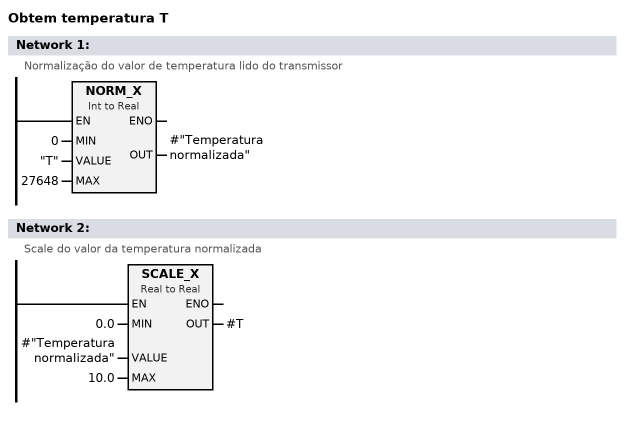
   RUNG wire#powerrail
      { S7_Templates := "[SrcType := Int, DestType := Real]" } Normalize(min := 0, value := "T", max := 27648, out => #"Temperatura normalizada")
   END_RUNG
   // the same network as SCL:
   #"Temperatura normalizada" := NORM_X(MIN := 0, VALUE := "T", MAX := 27648);
END_REGION

REGION Network 2
   // Scale do valor da temperatura normalizada
   RUNG wire#powerrail
      { S7_Templates := "[SrcType := Real, DestType := Real]" } Scale(min := 0.0, value := #"Temperatura normalizada", max := 10.0, out => #T)
   END_RUNG
   // the same network as SCL:
   #T := SCALE_X(MIN := 0.0, VALUE := #"Temperatura normalizada", MAX := 10.0);
END_REGION
END_FUNCTION

FUNCTION "Obtem temperatura TA" : Void   // FC23, LAD
{ S7_Optimized_Access := 'TRUE' }
VERSION : 0.1
   VAR_OUTPUT
      TA : Real;   // Temperatura obtida
   END_VAR
   VAR_TEMP
      "Temperatura normalizada" : Real;   // Temperatura normalizada
   END_VAR
BEGIN

REGION Network 1
   // Normalização do valor de temperatura lido do transmissor
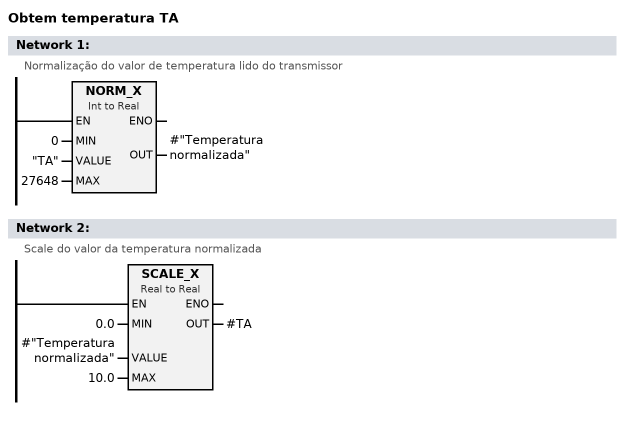
   RUNG wire#powerrail
      { S7_Templates := "[SrcType := Int, DestType := Real]" } Normalize(min := 0, value := "TA", max := 27648, out => #"Temperatura normalizada")
   END_RUNG
   // the same network as SCL:
   #"Temperatura normalizada" := NORM_X(MIN := 0, VALUE := "TA", MAX := 27648);
END_REGION

REGION Network 2
   // Scale do valor da temperatura normalizada
   RUNG wire#powerrail
      { S7_Templates := "[SrcType := Real, DestType := Real]" } Scale(min := 0.0, value := #"Temperatura normalizada", max := 10.0, out => #TA)
   END_RUNG
   // the same network as SCL:
   #TA := SCALE_X(MIN := 0.0, VALUE := #"Temperatura normalizada", MAX := 10.0);
END_REGION
END_FUNCTION

FUNCTION "Aciona VD2" : Void   // FC24, LAD
{ S7_Optimized_Access := 'TRUE' }
VERSION : 0.1
BEGIN

REGION Network 1: Válvula on/off da linha direta (segunda)
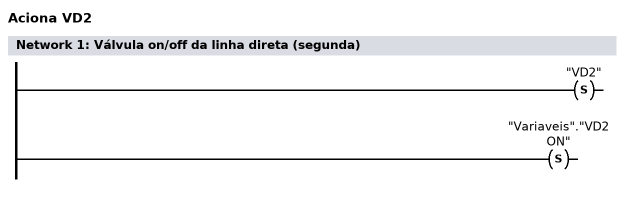
   RUNG wire#powerrail
      S_Coil( "VD2" )
   END_RUNG
   RUNG wire#powerrail
      S_Coil( "Variaveis"."VD2 ON" )
   END_RUNG
   // the same network as SCL:
   "VD2" := TRUE;
   "Variaveis"."VD2 ON" := TRUE;
END_REGION
END_FUNCTION

FUNCTION "Desliga VD2" : Void   // FC25, LAD
{ S7_Optimized_Access := 'TRUE' }
VERSION : 0.1
BEGIN

REGION Network 1: Válvula on/off da linha direta (segunda)
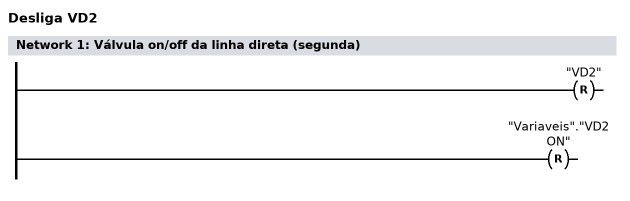
   RUNG wire#powerrail
      R_Coil( "VD2" )
   END_RUNG
   RUNG wire#powerrail
      R_Coil( "Variaveis"."VD2 ON" )
   END_RUNG
   // the same network as SCL:
   "VD2" := FALSE;
   "Variaveis"."VD2 ON" := FALSE;
END_REGION
END_FUNCTION

FUNCTION "Etapa pausada" : Void   // FC26, LAD
{ S7_Optimized_Access := 'TRUE' }
VERSION : 0.1
   VAR_TEMP   // added for the SCL form of the ladder/FBD networks
      _w1 : Bool;
      _w2 : Bool;
   END_VAR
BEGIN

REGION Network 1: LED que indica o estado de etapa pausada
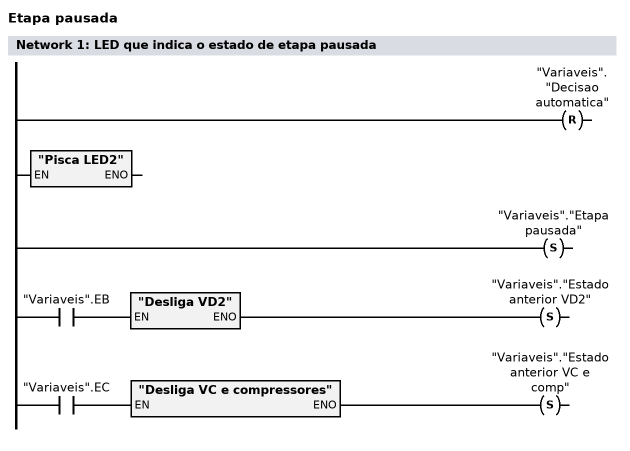
   RUNG wire#powerrail
      R_Coil( "Variaveis"."Decisao automatica" )
   END_RUNG
   RUNG wire#powerrail
      "Pisca LED2"()
   END_RUNG
   RUNG wire#powerrail
      S_Coil( "Variaveis"."Etapa pausada" )
   END_RUNG
   RUNG wire#powerrail
      Contact( "Variaveis".EB )
      "Desliga VD2"()
      S_Coil( "Variaveis"."Estado anterior VD2" )
   END_RUNG
   RUNG wire#powerrail
      Contact( "Variaveis".EC )
      "Desliga VC e compressores"()
      S_Coil( "Variaveis"."Estado anterior VC e comp" )
   END_RUNG
   // the same network as SCL:
   "Variaveis"."Decisao automatica" := FALSE;
   "Pisca LED2"();
   "Variaveis"."Etapa pausada" := TRUE;
   "Desliga VD2"(EN := "Variaveis".EB, ENO => #_w1);
   IF #_w1 THEN "Variaveis"."Estado anterior VD2" := TRUE; END_IF;
   "Desliga VC e compressores"(EN := "Variaveis".EC, ENO => #_w2);
   IF #_w2 THEN "Variaveis"."Estado anterior VC e comp" := TRUE; END_IF;
END_REGION
END_FUNCTION

FUNCTION "Etapa retomada" : Void   // FC27, LAD
{ S7_Optimized_Access := 'TRUE' }
VERSION : 0.1
BEGIN

REGION Network 1: LED que indica o estado de etapa pausada
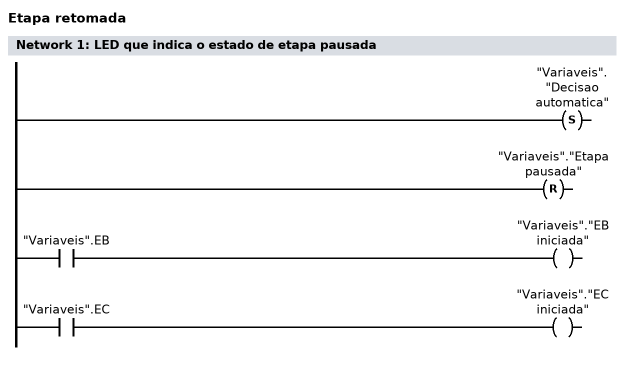
   RUNG wire#powerrail
      S_Coil( "Variaveis"."Decisao automatica" )
   END_RUNG
   RUNG wire#powerrail
      R_Coil( "Variaveis"."Etapa pausada" )
   END_RUNG
   RUNG wire#powerrail
      Contact( "Variaveis".EB )
      Coil( "Variaveis"."EB iniciada" )
   END_RUNG
   RUNG wire#powerrail
      Contact( "Variaveis".EC )
      Coil( "Variaveis"."EC iniciada" )
   END_RUNG
   // the same network as SCL:
   "Variaveis"."Decisao automatica" := TRUE;
   "Variaveis"."Etapa pausada" := FALSE;
   "Variaveis"."EB iniciada" := "Variaveis".EB;
   "Variaveis"."EC iniciada" := "Variaveis".EC;
END_REGION
END_FUNCTION

FUNCTION "Verifica VC 1" : Void   // FC28, LAD
{ S7_Optimized_Access := 'TRUE' }
VERSION : 0.1
BEGIN

REGION Network 1: Válvula on/off da entrada do sistema de compressores
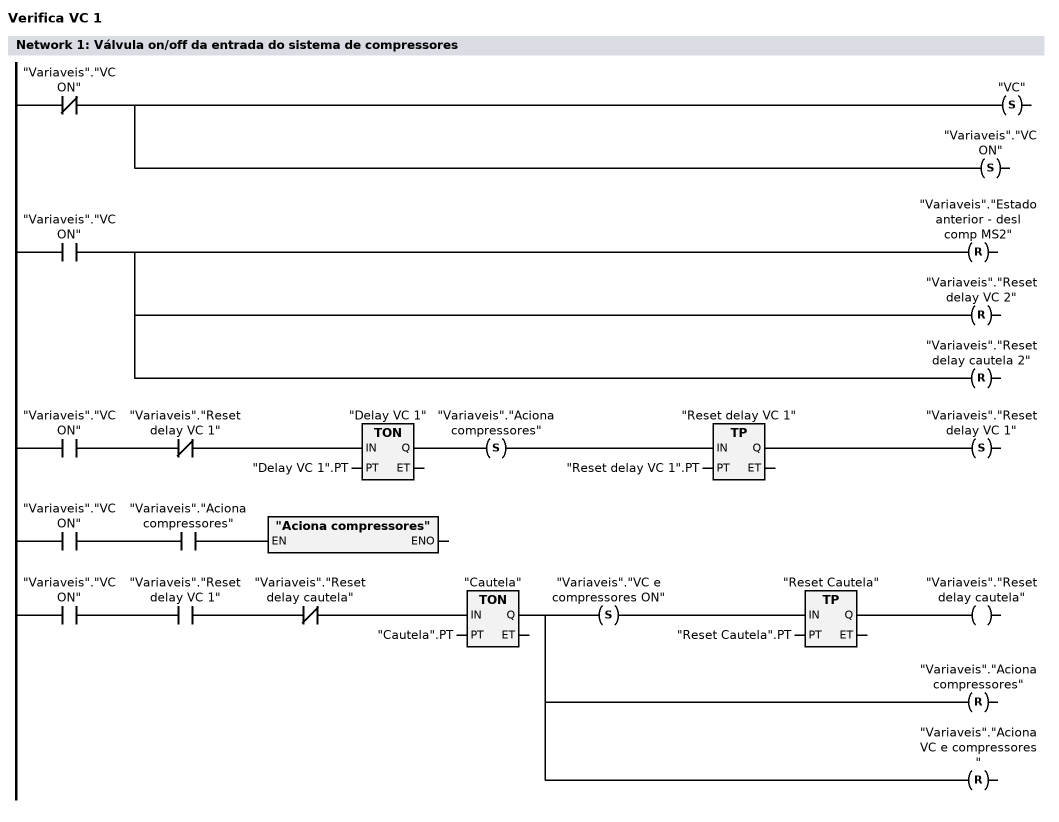
   IF NOT "Variaveis"."VC ON" THEN
       "VC" := TRUE;
       "Variaveis"."VC ON" := TRUE;
   END_IF;
   IF "Variaveis"."VC ON" THEN
       "Variaveis"."Estado anterior - desl comp MS2" := FALSE;
       "Variaveis"."Reset delay VC 2" := FALSE;
       "Variaveis"."Reset delay cautela 2" := FALSE;
   END_IF;
   "Delay VC 1".TON(IN := "Variaveis"."VC ON" AND NOT "Variaveis"."Reset delay VC 1", PT := "Delay VC 1".PT);
   IF "Delay VC 1".Q THEN "Variaveis"."Aciona compressores" := TRUE; END_IF;
   "Reset delay VC 1".TP(IN := "Delay VC 1".Q, PT := "Reset delay VC 1".PT);
   IF "Reset delay VC 1".Q THEN "Variaveis"."Reset delay VC 1" := TRUE; END_IF;
   IF "Variaveis"."VC ON" AND "Variaveis"."Aciona compressores" THEN "Aciona compressores"(); END_IF;
   "Cautela".TON(IN := "Variaveis"."VC ON" AND "Variaveis"."Reset delay VC 1" AND NOT "Variaveis"."Reset delay cautela",
                 PT := "Cautela".PT);
   IF "Cautela".Q THEN "Variaveis"."VC e compressores ON" := TRUE; END_IF;
   "Reset Cautela".TP(IN := "Cautela".Q, PT := "Reset Cautela".PT);
   "Variaveis"."Reset delay cautela" := "Reset Cautela".Q;
   IF "Cautela".Q THEN
       "Variaveis"."Aciona compressores" := FALSE;
       "Variaveis"."Aciona VC e compressores" := FALSE;
   END_IF;
END_REGION
END_FUNCTION

FUNCTION "Verifica VC 2" : Void   // FC29, LAD
{ S7_Optimized_Access := 'TRUE' }
VERSION : 0.1
BEGIN

REGION Network 1: Válvula on/off da entrada do sistema de compressores
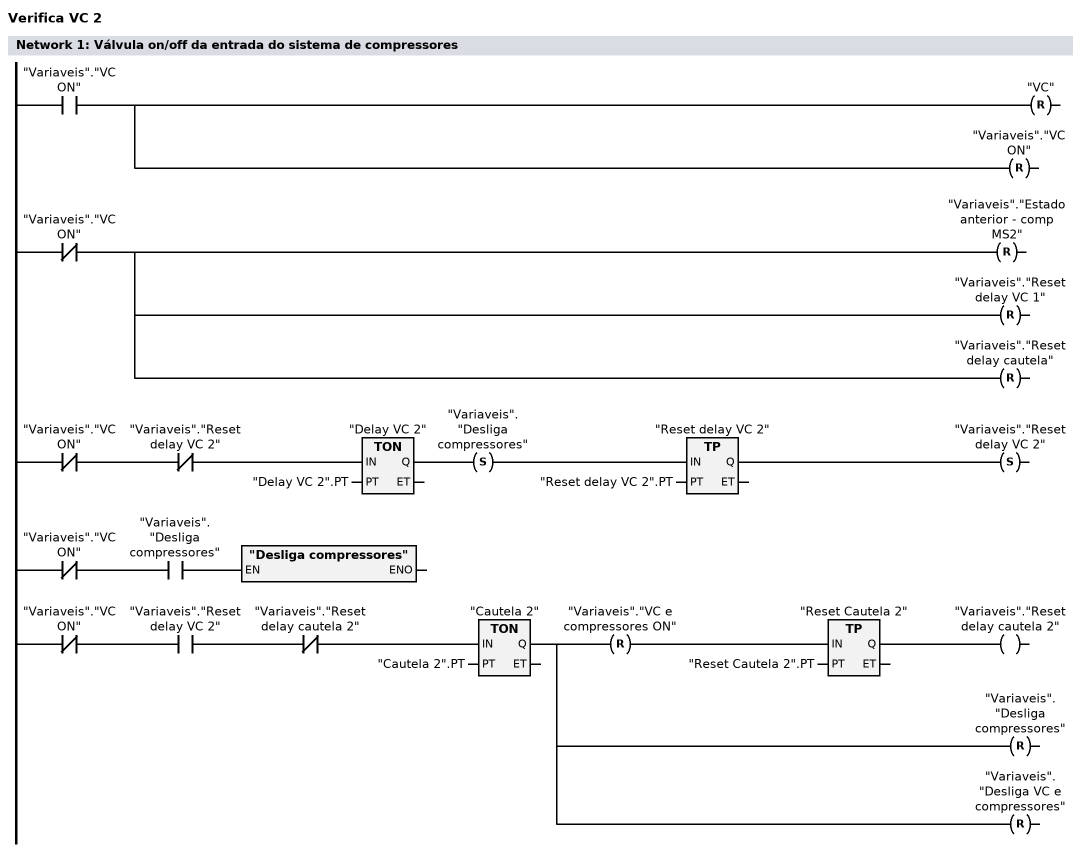
   IF "Variaveis"."VC ON" THEN
       "VC" := FALSE;
       "Variaveis"."VC ON" := FALSE;
   END_IF;
   IF NOT "Variaveis"."VC ON" THEN
       "Variaveis"."Estado anterior - comp MS2" := FALSE;
       "Variaveis"."Reset delay VC 1" := FALSE;
       "Variaveis"."Reset delay cautela" := FALSE;
   END_IF;
   "Delay VC 2".TON(IN := NOT "Variaveis"."VC ON" AND NOT "Variaveis"."Reset delay VC 2", PT := "Delay VC 2".PT);
   IF "Delay VC 2".Q THEN "Variaveis"."Desliga compressores" := TRUE; END_IF;
   "Reset delay VC 2".TP(IN := "Delay VC 2".Q, PT := "Reset delay VC 2".PT);
   IF "Reset delay VC 2".Q THEN "Variaveis"."Reset delay VC 2" := TRUE; END_IF;
   IF NOT "Variaveis"."VC ON" AND "Variaveis"."Desliga compressores" THEN "Desliga compressores"(); END_IF;
   "Cautela 2".TON(IN := NOT "Variaveis"."VC ON" AND "Variaveis"."Reset delay VC 2" AND NOT "Variaveis"."Reset delay cautela 2",
                   PT := "Cautela 2".PT);
   IF "Cautela 2".Q THEN "Variaveis"."VC e compressores ON" := FALSE; END_IF;
   "Reset Cautela 2".TP(IN := "Cautela 2".Q, PT := "Reset Cautela 2".PT);
   "Variaveis"."Reset delay cautela 2" := "Reset Cautela 2".Q;
   IF "Cautela 2".Q THEN
       "Variaveis"."Desliga compressores" := FALSE;
       "Variaveis"."Desliga VC e compressores" := FALSE;
   END_IF;
END_REGION
END_FUNCTION

FUNCTION "Aciona VC e compressores" : Void   // FC30, LAD
{ S7_Optimized_Access := 'TRUE' }
VERSION : 0.1
BEGIN

REGION Network 1
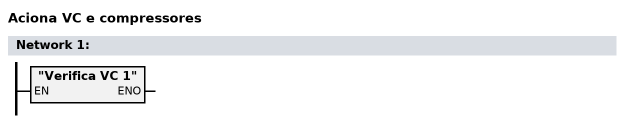
   RUNG wire#powerrail
      "Verifica VC 1"()
   END_RUNG
   // the same network as SCL:
   "Verifica VC 1"();
END_REGION
END_FUNCTION

FUNCTION "Desliga VC e compressores" : Void   // FC31, LAD
{ S7_Optimized_Access := 'TRUE' }
VERSION : 0.1
BEGIN

REGION Network 1
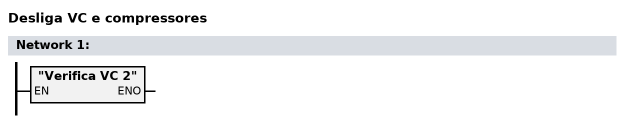
   RUNG wire#powerrail
      "Verifica VC 2"()
   END_RUNG
   // the same network as SCL:
   "Verifica VC 2"();
END_REGION
END_FUNCTION

FUNCTION "EB - Etapa iniciada" : Void   // FC32, LAD
{ S7_Optimized_Access := 'TRUE' }
VERSION : 0.1
   VAR_TEMP
      T : Real;   // Temperatura no nó estendido
      TA : Real;   // Temperatura ambiente
      PN : Real;   // Pressão no nó estendido
      PSF6 : Real;   // Pressão do tanque de SF6
      "Threshold ambiente" : Real;   // (1 - beta)*TA
      "Threshold PSF6" : Real;   // (1 + gamma)*PSF6
   END_VAR
   VAR_TEMP   // added for the SCL form of the ladder/FBD networks
      _w1 : Bool;
      _w2 : Bool;
      _w3 : Bool;
      _w4 : Bool;
   END_VAR
BEGIN

REGION Network 1
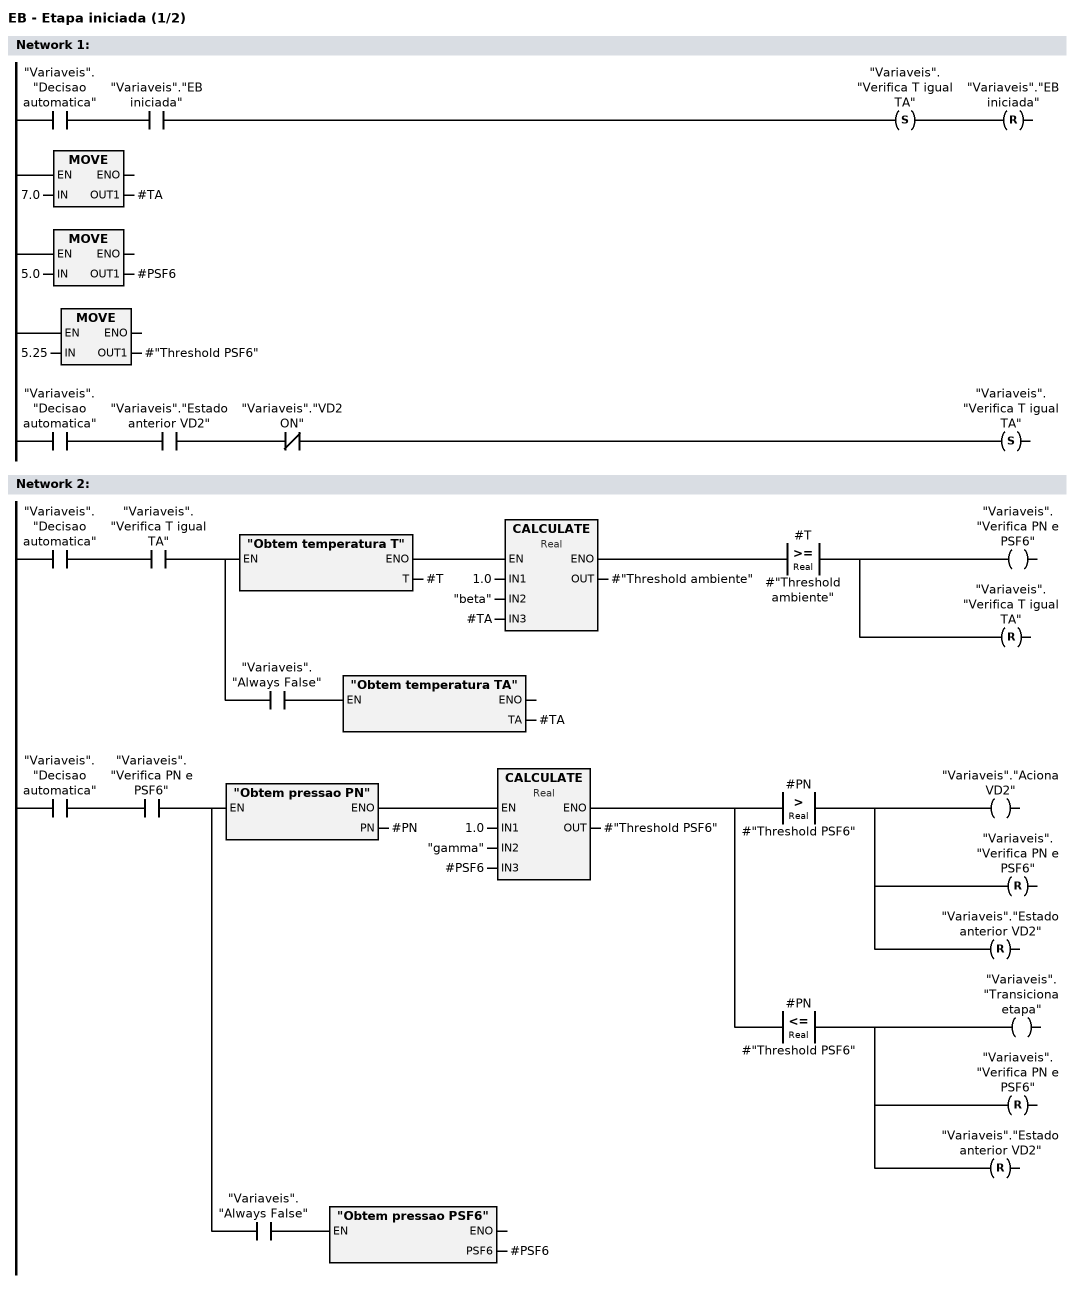
   RUNG wire#powerrail
      Contact( "Variaveis"."Decisao automatica" )
      Contact( "Variaveis"."EB iniciada" )
      S_Coil( "Variaveis"."Verifica T igual TA" )
      R_Coil( "Variaveis"."EB iniciada" )
   END_RUNG
   RUNG wire#powerrail
      Move(in := 7.0, out1 => #TA)
   END_RUNG
   RUNG wire#powerrail
      Move(in := 5.0, out1 => #PSF6)
   END_RUNG
   RUNG wire#powerrail
      Move(in := 5.25, out1 => #"Threshold PSF6")
   END_RUNG
   RUNG wire#powerrail
      Contact( "Variaveis"."Decisao automatica" )
      Contact( "Variaveis"."Estado anterior VD2" )
      I_Contact( "Variaveis"."VD2 ON" )
      S_Coil( "Variaveis"."Verifica T igual TA" )
   END_RUNG
   // the same network as SCL:
   IF "Variaveis"."Decisao automatica" AND "Variaveis"."EB iniciada" THEN
       "Variaveis"."Verifica T igual TA" := TRUE;
       "Variaveis"."EB iniciada" := FALSE;
   END_IF;
   #TA := 7.0;
   #PSF6 := 5.0;
   #"Threshold PSF6" := 5.25;
   IF "Variaveis"."Decisao automatica" AND "Variaveis"."Estado anterior VD2" AND NOT "Variaveis"."VD2 ON" THEN
       "Variaveis"."Verifica T igual TA" := TRUE;
   END_IF;
END_REGION

REGION Network 2
   RUNG wire#powerrail
      Contact( "Variaveis"."Decisao automatica" )
      Contact( "Variaveis"."Verifica T igual TA" )
      wire#w1
      "Obtem temperatura T"(T => #T)
      { S7_Templates := "SrcType := Real"; S7_Expression := "(IN1 - IN2) * IN3" } Calculate(in1 := 1.0, in2 := "beta", in3 := #TA, out => #"Threshold ambiente")
      { S7_Templates := "SrcType := Real" } GE_Contact(in1 := #T, in2 := #"Threshold ambiente")
      wire#w2
      Coil( "Variaveis"."Verifica PN e PSF6" )
   END_RUNG
   RUNG wire#w2
      R_Coil( "Variaveis"."Verifica T igual TA" )
   END_RUNG
   RUNG wire#w1
      Contact( "Variaveis"."Always False" )
      "Obtem temperatura TA"(TA => #TA)
   END_RUNG
   RUNG wire#powerrail
      Contact( "Variaveis"."Decisao automatica" )
      Contact( "Variaveis"."Verifica PN e PSF6" )
      wire#w3
      "Obtem pressao PN"(PN => #PN)
      { S7_Templates := "SrcType := Real"; S7_Expression := "(IN1 + IN2) * IN3" } Calculate(in1 := 1.0, in2 := "gamma", in3 := #PSF6, out => #"Threshold PSF6")
      wire#w4
      { S7_Templates := "SrcType := Real" } GT_Contact(in1 := #PN, in2 := #"Threshold PSF6")
      wire#w5
      Coil( "Variaveis"."Aciona VD2" )
   END_RUNG
   RUNG wire#w5
      R_Coil( "Variaveis"."Verifica PN e PSF6" )
   END_RUNG
   RUNG wire#w5
      R_Coil( "Variaveis"."Estado anterior VD2" )
   END_RUNG
   RUNG wire#w4
      { S7_Templates := "SrcType := Real" } LE_Contact(in1 := #PN, in2 := #"Threshold PSF6")
      wire#w6
      Coil( "Variaveis"."Transiciona etapa" )
   END_RUNG
   RUNG wire#w6
      R_Coil( "Variaveis"."Verifica PN e PSF6" )
   END_RUNG
   RUNG wire#w6
      R_Coil( "Variaveis"."Estado anterior VD2" )
   END_RUNG
   RUNG wire#w3
      Contact( "Variaveis"."Always False" )
      "Obtem pressao PSF6"(PSF6 => #PSF6)
   END_RUNG
   // the same network as SCL:
   #_w1 := "Variaveis"."Decisao automatica" AND "Variaveis"."Verifica T igual TA";
   "Obtem temperatura T"(EN := #_w1, T => #T, ENO => #_w2);
   IF #_w2 THEN #"Threshold ambiente" := (1.0 - "beta") * #TA; END_IF;
   "Variaveis"."Verifica PN e PSF6" := #_w2 AND (#T >= #"Threshold ambiente");
   IF "Variaveis"."Verifica PN e PSF6" THEN "Variaveis"."Verifica T igual TA" := FALSE; END_IF;
   IF #_w1 AND "Variaveis"."Always False" THEN "Obtem temperatura TA"(TA => #TA); END_IF;
   #_w3 := "Variaveis"."Decisao automatica" AND "Variaveis"."Verifica PN e PSF6";
   "Obtem pressao PN"(EN := #_w3, PN => #PN, ENO => #_w4);
   IF #_w4 THEN #"Threshold PSF6" := (1.0 + "gamma") * #PSF6; END_IF;
   "Variaveis"."Aciona VD2" := #_w4 AND (#PN > #"Threshold PSF6");
   IF "Variaveis"."Aciona VD2" THEN
       "Variaveis"."Verifica PN e PSF6" := FALSE;
       "Variaveis"."Estado anterior VD2" := FALSE;
   END_IF;
   "Variaveis"."Transiciona etapa" := #_w4 AND (#PN <= #"Threshold PSF6");
   IF "Variaveis"."Transiciona etapa" THEN
       "Variaveis"."Verifica PN e PSF6" := FALSE;
       "Variaveis"."Estado anterior VD2" := FALSE;
   END_IF;
   IF #_w3 AND "Variaveis"."Always False" THEN "Obtem pressao PSF6"(PSF6 => #PSF6); END_IF;
END_REGION

REGION Network 3
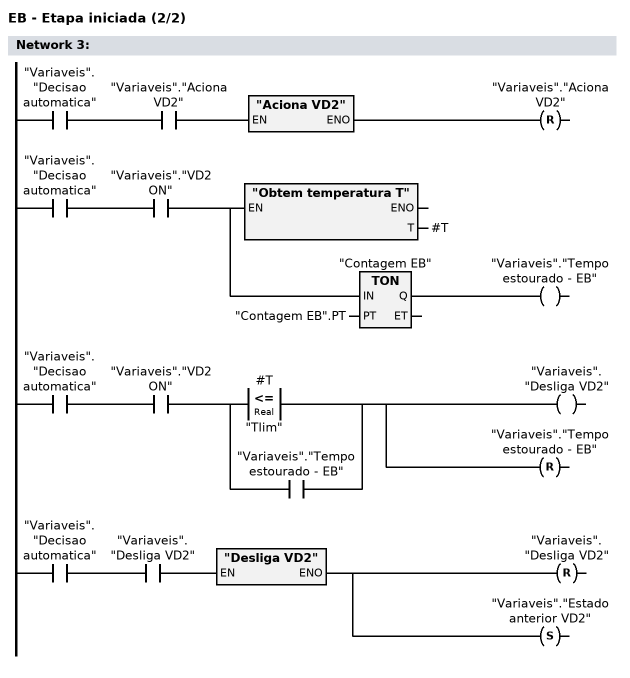
   "Aciona VD2"(EN := "Variaveis"."Decisao automatica" AND "Variaveis"."Aciona VD2", ENO => #_w1);
   IF #_w1 THEN "Variaveis"."Aciona VD2" := FALSE; END_IF;
   #_w2 := "Variaveis"."Decisao automatica" AND "Variaveis"."VD2 ON";
   IF #_w2 THEN "Obtem temperatura T"(T => #T); END_IF;
   "Contagem EB".TON(IN := #_w2, PT := "Contagem EB".PT);
   "Variaveis"."Tempo estourado - EB" := "Contagem EB".Q;
   "Variaveis"."Desliga VD2" := "Variaveis"."Decisao automatica" AND "Variaveis"."VD2 ON" AND ((#T <= "Tlim") OR "Variaveis"."Tempo estourado - EB");
   IF "Variaveis"."Desliga VD2" THEN "Variaveis"."Tempo estourado - EB" := FALSE; END_IF;
   "Desliga VD2"(EN := "Variaveis"."Decisao automatica" AND "Variaveis"."Desliga VD2", ENO => #_w3);
   IF #_w3 THEN
       "Variaveis"."Desliga VD2" := FALSE;
       "Variaveis"."Estado anterior VD2" := TRUE;
   END_IF;
END_REGION
END_FUNCTION

FUNCTION "EB - Etapa finalizada" : Void   // FC33, LAD
{ S7_Optimized_Access := 'TRUE' }
VERSION : 0.1
BEGIN

REGION Network 1
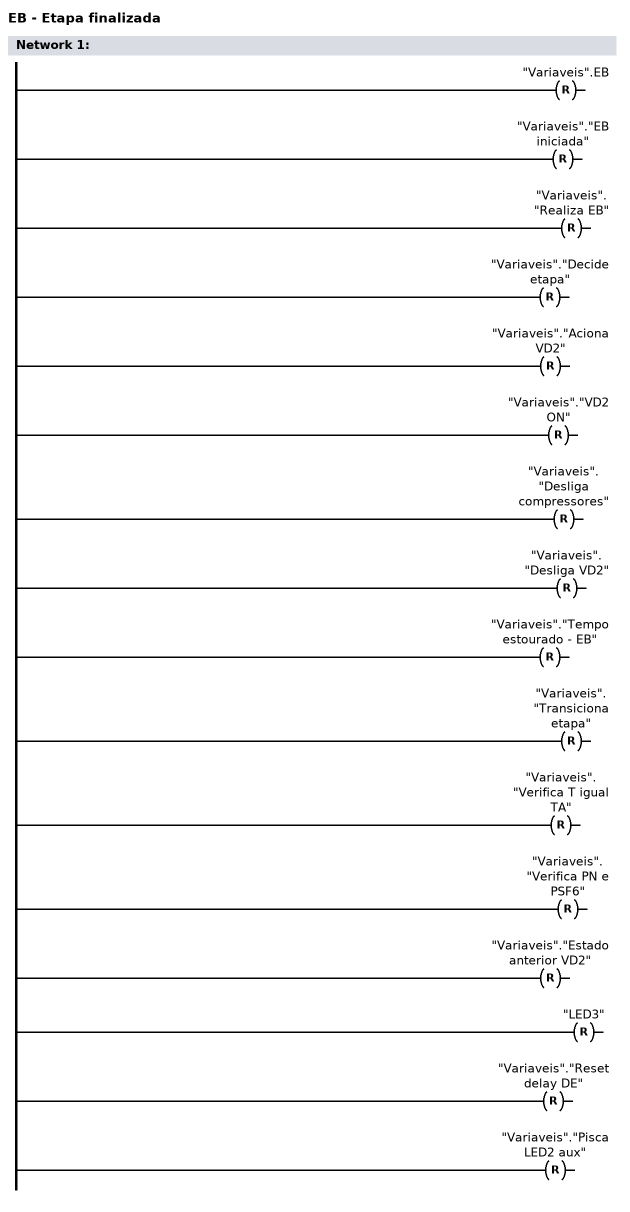
   RUNG wire#powerrail
      R_Coil( "Variaveis".EB )
   END_RUNG
   RUNG wire#powerrail
      R_Coil( "Variaveis"."EB iniciada" )
   END_RUNG
   RUNG wire#powerrail
      R_Coil( "Variaveis"."Realiza EB" )
   END_RUNG
   RUNG wire#powerrail
      R_Coil( "Variaveis"."Decide etapa" )
   END_RUNG
   RUNG wire#powerrail
      R_Coil( "Variaveis"."Aciona VD2" )
   END_RUNG
   RUNG wire#powerrail
      R_Coil( "Variaveis"."VD2 ON" )
   END_RUNG
   RUNG wire#powerrail
      R_Coil( "Variaveis"."Desliga compressores" )
   END_RUNG
   RUNG wire#powerrail
      R_Coil( "Variaveis"."Desliga VD2" )
   END_RUNG
   RUNG wire#powerrail
      R_Coil( "Variaveis"."Tempo estourado - EB" )
   END_RUNG
   RUNG wire#powerrail
      R_Coil( "Variaveis"."Transiciona etapa" )
   END_RUNG
   RUNG wire#powerrail
      R_Coil( "Variaveis"."Verifica T igual TA" )
   END_RUNG
   RUNG wire#powerrail
      R_Coil( "Variaveis"."Verifica PN e PSF6" )
   END_RUNG
   RUNG wire#powerrail
      R_Coil( "Variaveis"."Estado anterior VD2" )
   END_RUNG
   RUNG wire#powerrail
      R_Coil( "LED3" )
   END_RUNG
   RUNG wire#powerrail
      R_Coil( "Variaveis"."Reset delay DE" )
   END_RUNG
   RUNG wire#powerrail
      R_Coil( "Variaveis"."Pisca LED2 aux" )
   END_RUNG
   // the same network as SCL:
   "Variaveis".EB := FALSE;
   "Variaveis"."EB iniciada" := FALSE;
   "Variaveis"."Realiza EB" := FALSE;
   "Variaveis"."Decide etapa" := FALSE;
   "Variaveis"."Aciona VD2" := FALSE;
   "Variaveis"."VD2 ON" := FALSE;
   "Variaveis"."Desliga compressores" := FALSE;
   "Variaveis"."Desliga VD2" := FALSE;
   "Variaveis"."Tempo estourado - EB" := FALSE;
   "Variaveis"."Transiciona etapa" := FALSE;
   "Variaveis"."Verifica T igual TA" := FALSE;
   "Variaveis"."Verifica PN e PSF6" := FALSE;
   "Variaveis"."Estado anterior VD2" := FALSE;
   "LED3" := FALSE;
   "Variaveis"."Reset delay DE" := FALSE;
   "Variaveis"."Pisca LED2 aux" := FALSE;
END_REGION
END_FUNCTION

FUNCTION "EC - Etapa iniciada" : Void   // FC34, LAD
{ S7_Optimized_Access := 'TRUE' }
VERSION : 0.1
   VAR_TEMP
      T : Real;   // Temperatura no nó estendido
      TA : Real;   // Temperatura ambiente
      PN : Real;   // Pressão no nó estendido
      PSF6 : Real;   // Pressão do tanque de SF6
      "Threshold ambiente" : Real;   // (1 - beta)*TA
   END_VAR
   VAR_TEMP   // added for the SCL form of the ladder/FBD networks
      _w1 : Bool;
      _w2 : Bool;
      _w3 : Bool;
   END_VAR
BEGIN

REGION Network 1
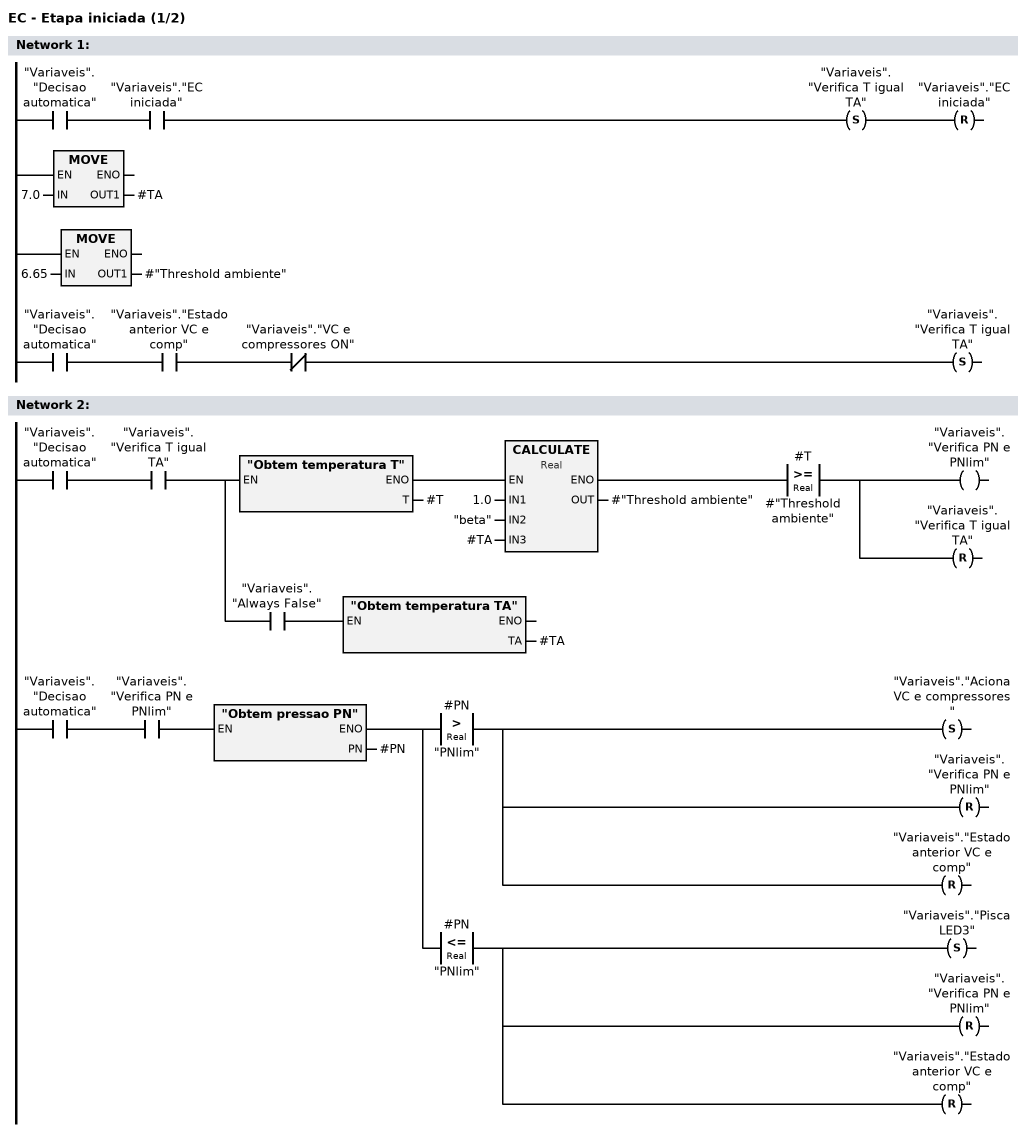
   RUNG wire#powerrail
      Contact( "Variaveis"."Decisao automatica" )
      Contact( "Variaveis"."EC iniciada" )
      S_Coil( "Variaveis"."Verifica T igual TA" )
      R_Coil( "Variaveis"."EC iniciada" )
   END_RUNG
   RUNG wire#powerrail
      Move(in := 7.0, out1 => #TA)
   END_RUNG
   RUNG wire#powerrail
      Move(in := 6.65, out1 => #"Threshold ambiente")
   END_RUNG
   RUNG wire#powerrail
      Contact( "Variaveis"."Decisao automatica" )
      Contact( "Variaveis"."Estado anterior VC e comp" )
      I_Contact( "Variaveis"."VC e compressores ON" )
      S_Coil( "Variaveis"."Verifica T igual TA" )
   END_RUNG
   // the same network as SCL:
   IF "Variaveis"."Decisao automatica" AND "Variaveis"."EC iniciada" THEN
       "Variaveis"."Verifica T igual TA" := TRUE;
       "Variaveis"."EC iniciada" := FALSE;
   END_IF;
   #TA := 7.0;
   #"Threshold ambiente" := 6.65;
   IF "Variaveis"."Decisao automatica" AND "Variaveis"."Estado anterior VC e comp" AND NOT "Variaveis"."VC e compressores ON" THEN
       "Variaveis"."Verifica T igual TA" := TRUE;
   END_IF;
END_REGION

REGION Network 2
   RUNG wire#powerrail
      Contact( "Variaveis"."Decisao automatica" )
      Contact( "Variaveis"."Verifica T igual TA" )
      wire#w1
      "Obtem temperatura T"(T => #T)
      { S7_Templates := "SrcType := Real"; S7_Expression := "(IN1 - IN2) * IN3" } Calculate(in1 := 1.0, in2 := "beta", in3 := #TA, out => #"Threshold ambiente")
      { S7_Templates := "SrcType := Real" } GE_Contact(in1 := #T, in2 := #"Threshold ambiente")
      wire#w2
      Coil( "Variaveis"."Verifica PN e PNlim" )
   END_RUNG
   RUNG wire#w2
      R_Coil( "Variaveis"."Verifica T igual TA" )
   END_RUNG
   RUNG wire#w1
      Contact( "Variaveis"."Always False" )
      "Obtem temperatura TA"(TA => #TA)
   END_RUNG
   RUNG wire#powerrail
      Contact( "Variaveis"."Decisao automatica" )
      Contact( "Variaveis"."Verifica PN e PNlim" )
      "Obtem pressao PN"(PN => #PN)
      wire#w3
      { S7_Templates := "SrcType := Real" } GT_Contact(in1 := #PN, in2 := "PNlim")
      wire#w4
      S_Coil( "Variaveis"."Aciona VC e compressores" )
   END_RUNG
   RUNG wire#w4
      R_Coil( "Variaveis"."Verifica PN e PNlim" )
   END_RUNG
   RUNG wire#w4
      R_Coil( "Variaveis"."Estado anterior VC e comp" )
   END_RUNG
   RUNG wire#w3
      { S7_Templates := "SrcType := Real" } LE_Contact(in1 := #PN, in2 := "PNlim")
      wire#w5
      S_Coil( "Variaveis"."Pisca LED3" )
   END_RUNG
   RUNG wire#w5
      R_Coil( "Variaveis"."Verifica PN e PNlim" )
   END_RUNG
   RUNG wire#w5
      R_Coil( "Variaveis"."Estado anterior VC e comp" )
   END_RUNG
   // the same network as SCL:
   #_w1 := "Variaveis"."Decisao automatica" AND "Variaveis"."Verifica T igual TA";
   "Obtem temperatura T"(EN := #_w1, T => #T, ENO => #_w2);
   IF #_w2 THEN #"Threshold ambiente" := (1.0 - "beta") * #TA; END_IF;
   "Variaveis"."Verifica PN e PNlim" := #_w2 AND (#T >= #"Threshold ambiente");
   IF "Variaveis"."Verifica PN e PNlim" THEN "Variaveis"."Verifica T igual TA" := FALSE; END_IF;
   IF #_w1 AND "Variaveis"."Always False" THEN "Obtem temperatura TA"(TA => #TA); END_IF;
   "Obtem pressao PN"(EN := "Variaveis"."Decisao automatica" AND "Variaveis"."Verifica PN e PNlim",
                      PN => #PN,
                      ENO => #_w3);
   IF #_w3 AND (#PN > "PNlim") THEN
       "Variaveis"."Aciona VC e compressores" := TRUE;
       "Variaveis"."Verifica PN e PNlim" := FALSE;
       "Variaveis"."Estado anterior VC e comp" := FALSE;
   END_IF;
   IF #_w3 AND (#PN <= "PNlim") THEN
       "Variaveis"."Pisca LED3" := TRUE;
       "Variaveis"."Verifica PN e PNlim" := FALSE;
       "Variaveis"."Estado anterior VC e comp" := FALSE;
   END_IF;
END_REGION

REGION Network 3
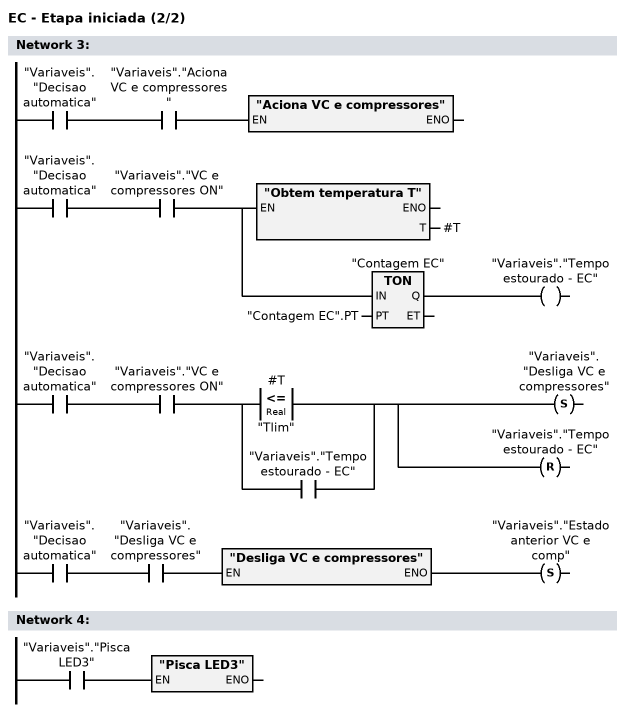
   IF "Variaveis"."Decisao automatica" AND "Variaveis"."Aciona VC e compressores" THEN
       "Aciona VC e compressores"();
   END_IF;
   #_w1 := "Variaveis"."Decisao automatica" AND "Variaveis"."VC e compressores ON";
   IF #_w1 THEN "Obtem temperatura T"(T => #T); END_IF;
   "Contagem EC".TON(IN := #_w1, PT := "Contagem EC".PT);
   "Variaveis"."Tempo estourado - EC" := "Contagem EC".Q;
   IF "Variaveis"."Decisao automatica" AND "Variaveis"."VC e compressores ON" AND ((#T <= "Tlim") OR "Variaveis"."Tempo estourado - EC") THEN
       "Variaveis"."Desliga VC e compressores" := TRUE;
       "Variaveis"."Tempo estourado - EC" := FALSE;
   END_IF;
   "Desliga VC e compressores"(EN := "Variaveis"."Decisao automatica" AND "Variaveis"."Desliga VC e compressores",
                           ENO => #_w2);
   IF #_w2 THEN "Variaveis"."Estado anterior VC e comp" := TRUE; END_IF;
END_REGION

REGION Network 4
   RUNG wire#powerrail
      Contact( "Variaveis"."Pisca LED3" )
      "Pisca LED3"()
   END_RUNG
   // the same network as SCL:
   IF "Variaveis"."Pisca LED3" THEN "Pisca LED3"(); END_IF;
END_REGION
END_FUNCTION

FUNCTION "EC - Etapa finalizada" : Void   // FC35, LAD
{ S7_Optimized_Access := 'TRUE' }
VERSION : 0.1
BEGIN

REGION Network 1
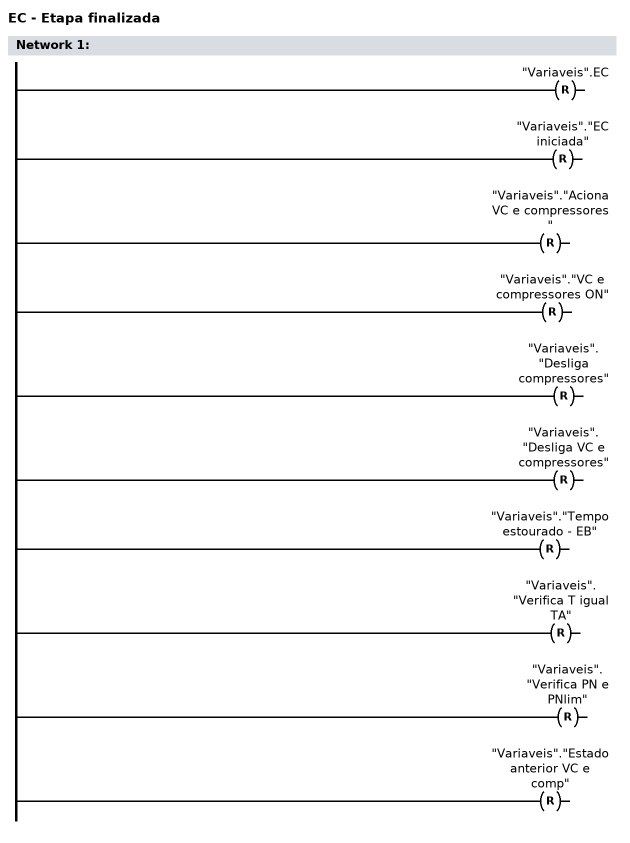
   RUNG wire#powerrail
      R_Coil( "Variaveis".EC )
   END_RUNG
   RUNG wire#powerrail
      R_Coil( "Variaveis"."EC iniciada" )
   END_RUNG
   RUNG wire#powerrail
      R_Coil( "Variaveis"."Aciona VC e compressores" )
   END_RUNG
   RUNG wire#powerrail
      R_Coil( "Variaveis"."VC e compressores ON" )
   END_RUNG
   RUNG wire#powerrail
      R_Coil( "Variaveis"."Desliga compressores" )
   END_RUNG
   RUNG wire#powerrail
      R_Coil( "Variaveis"."Desliga VC e compressores" )
   END_RUNG
   RUNG wire#powerrail
      R_Coil( "Variaveis"."Tempo estourado - EB" )
   END_RUNG
   RUNG wire#powerrail
      R_Coil( "Variaveis"."Verifica T igual TA" )
   END_RUNG
   RUNG wire#powerrail
      R_Coil( "Variaveis"."Verifica PN e PNlim" )
   END_RUNG
   RUNG wire#powerrail
      R_Coil( "Variaveis"."Estado anterior VC e comp" )
   END_RUNG
   // the same network as SCL:
   "Variaveis".EC := FALSE;
   "Variaveis"."EC iniciada" := FALSE;
   "Variaveis"."Aciona VC e compressores" := FALSE;
   "Variaveis"."VC e compressores ON" := FALSE;
   "Variaveis"."Desliga compressores" := FALSE;
   "Variaveis"."Desliga VC e compressores" := FALSE;
   "Variaveis"."Tempo estourado - EB" := FALSE;
   "Variaveis"."Verifica T igual TA" := FALSE;
   "Variaveis"."Verifica PN e PNlim" := FALSE;
   "Variaveis"."Estado anterior VC e comp" := FALSE;
END_REGION
END_FUNCTION

FUNCTION "MS2 - Operacao iniciada" : Void   // FC36, LAD
{ S7_Optimized_Access := 'TRUE' }
VERSION : 0.1
   VAR_TEMP
      PN : Real;   // Pressão no nó estendido
      PSF6 : Real;   // Pressão do tanque de SF6
      "Threshold PSF6" : Real;   // (1 + gamma)*PSF6
   END_VAR
   VAR_TEMP   // added for the SCL form of the ladder/FBD networks
      _w1 : Bool;
      _w2 : Bool;
      _w3 : Bool;
      _w4 : Bool;
   END_VAR
BEGIN

REGION Network 1: Válvula on/off da linha direta (primeira)
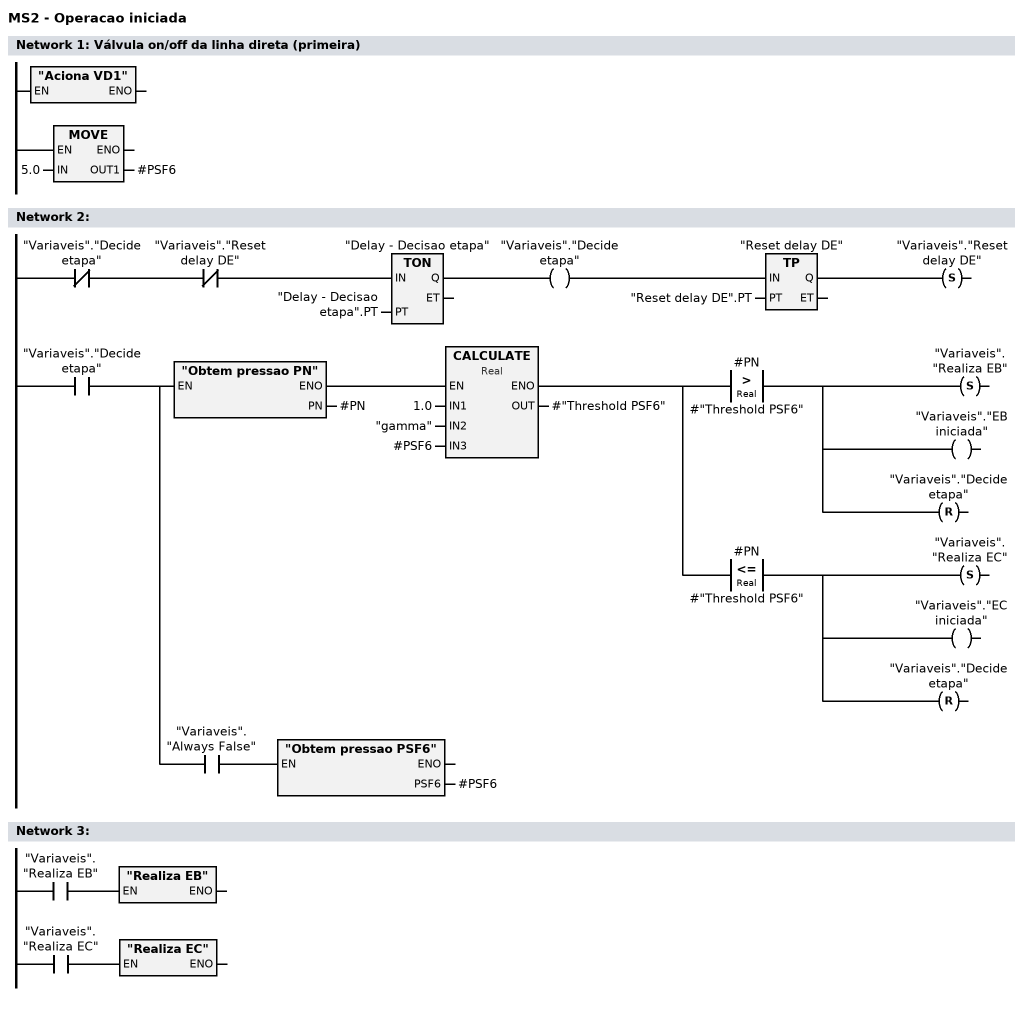
   RUNG wire#powerrail
      "Aciona VD1"()
   END_RUNG
   RUNG wire#powerrail
      Move(in := 5.0, out1 => #PSF6)
   END_RUNG
   // the same network as SCL:
   "Aciona VD1"();
   #PSF6 := 5.0;
END_REGION

REGION Network 2
   "Delay - Decisao etapa".TON(IN := NOT "Variaveis"."Decide etapa" AND NOT "Variaveis"."Reset delay DE",
                           PT := "Delay - Decisao etapa".PT);
   "Variaveis"."Decide etapa" := "Delay - Decisao etapa".Q;
   "Reset delay DE".TP(IN := "Delay - Decisao etapa".Q, PT := "Reset delay DE".PT);
   IF "Reset delay DE".Q THEN "Variaveis"."Reset delay DE" := TRUE; END_IF;
   #_w2 := "Variaveis"."Decide etapa";
   "Obtem pressao PN"(EN := "Variaveis"."Decide etapa", PN => #PN, ENO => #_w1);
   IF #_w1 THEN #"Threshold PSF6" := (1.0 + "gamma") * #PSF6; END_IF;
   #_w3 := #_w1 AND (#PN > #"Threshold PSF6");
   IF #_w3 THEN "Variaveis"."Realiza EB" := TRUE; END_IF;
   "Variaveis"."EB iniciada" := #_w3;
   IF #_w3 THEN "Variaveis"."Decide etapa" := FALSE; END_IF;
   #_w4 := #_w1 AND (#PN <= #"Threshold PSF6");
   IF #_w4 THEN "Variaveis"."Realiza EC" := TRUE; END_IF;
   "Variaveis"."EC iniciada" := #_w4;
   IF #_w4 THEN "Variaveis"."Decide etapa" := FALSE; END_IF;
   IF #_w2 AND "Variaveis"."Always False" THEN "Obtem pressao PSF6"(PSF6 => #PSF6); END_IF;
END_REGION

REGION Network 3
   RUNG wire#powerrail
      Contact( "Variaveis"."Realiza EB" )
      "Realiza EB"()
   END_RUNG
   RUNG wire#powerrail
      Contact( "Variaveis"."Realiza EC" )
      "Realiza EC"()
   END_RUNG
   // the same network as SCL:
   IF "Variaveis"."Realiza EB" THEN "Realiza EB"(); END_IF;
   IF "Variaveis"."Realiza EC" THEN "Realiza EC"(); END_IF;
END_REGION
END_FUNCTION

FUNCTION "Realiza EB" : Void   // FC37, LAD
{ S7_Optimized_Access := 'TRUE' }
VERSION : 0.1
   VAR_TEMP   // added for the SCL form of the ladder/FBD networks
      _w1 : Bool;
   END_VAR
BEGIN

REGION Network 1: LED que indica início/fim das etapas do MS2
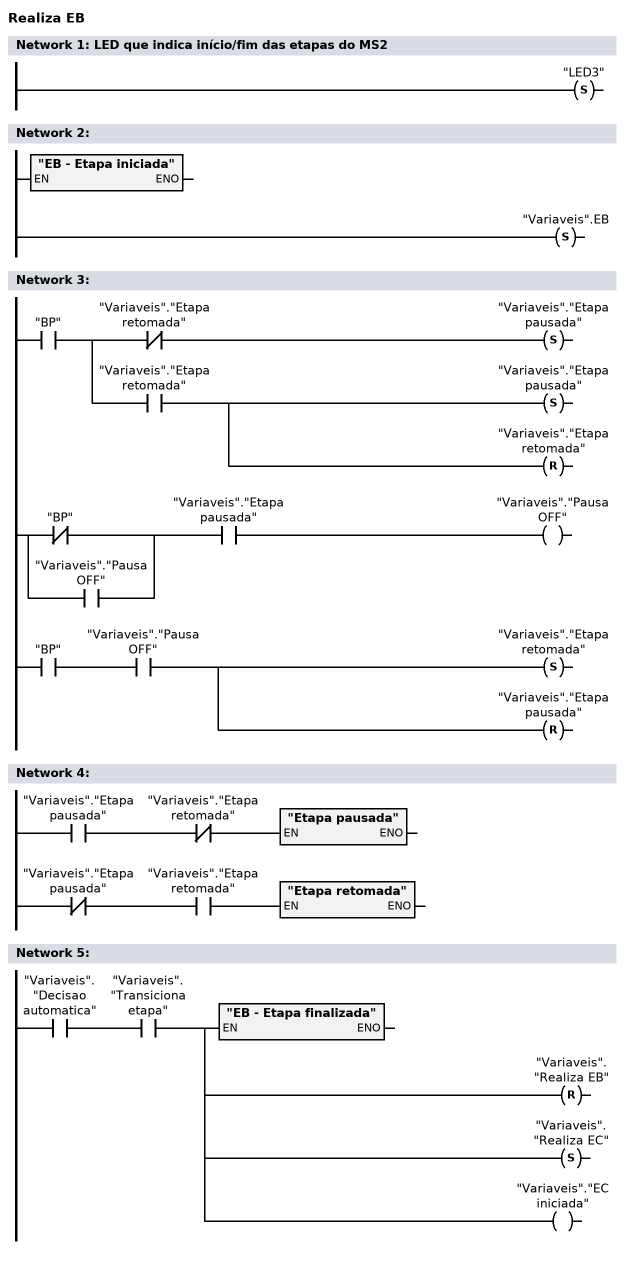
   RUNG wire#powerrail
      S_Coil( "LED3" )
   END_RUNG
   // the same network as SCL:
   "LED3" := TRUE;
END_REGION

REGION Network 2
   RUNG wire#powerrail
      "EB - Etapa iniciada"()
   END_RUNG
   RUNG wire#powerrail
      S_Coil( "Variaveis".EB )
   END_RUNG
   // the same network as SCL:
   "EB - Etapa iniciada"();
   "Variaveis".EB := TRUE;
END_REGION

REGION Network 3
   RUNG wire#powerrail
      Contact( "BP" )
      wire#w1
      I_Contact( "Variaveis"."Etapa retomada" )
      S_Coil( "Variaveis"."Etapa pausada" )
   END_RUNG
   RUNG wire#w1
      Contact( "Variaveis"."Etapa retomada" )
      wire#w2
      S_Coil( "Variaveis"."Etapa pausada" )
   END_RUNG
   RUNG wire#w2
      R_Coil( "Variaveis"."Etapa retomada" )
   END_RUNG
   RUNG wire#powerrail
      I_Contact( "BP" )
      wire#w3
      Contact( "Variaveis"."Etapa pausada" )
      Coil( "Variaveis"."Pausa OFF" )
   END_RUNG
   RUNG wire#powerrail
      Contact( "Variaveis"."Pausa OFF" )
   END_RUNG wire#w3
   RUNG wire#powerrail
      Contact( "BP" )
      Contact( "Variaveis"."Pausa OFF" )
      wire#w4
      S_Coil( "Variaveis"."Etapa retomada" )
   END_RUNG
   RUNG wire#w4
      R_Coil( "Variaveis"."Etapa pausada" )
   END_RUNG
   // the same network as SCL:
   IF "BP" AND NOT "Variaveis"."Etapa retomada" THEN "Variaveis"."Etapa pausada" := TRUE; END_IF;
   IF "BP" AND "Variaveis"."Etapa retomada" THEN
       "Variaveis"."Etapa pausada" := TRUE;
       "Variaveis"."Etapa retomada" := FALSE;
   END_IF;
   "Variaveis"."Pausa OFF" := (NOT "BP" OR "Variaveis"."Pausa OFF") AND "Variaveis"."Etapa pausada";
   IF "BP" AND "Variaveis"."Pausa OFF" THEN
       "Variaveis"."Etapa retomada" := TRUE;
       "Variaveis"."Etapa pausada" := FALSE;
   END_IF;
END_REGION

REGION Network 4
   RUNG wire#powerrail
      Contact( "Variaveis"."Etapa pausada" )
      I_Contact( "Variaveis"."Etapa retomada" )
      "Etapa pausada"()
   END_RUNG
   RUNG wire#powerrail
      I_Contact( "Variaveis"."Etapa pausada" )
      Contact( "Variaveis"."Etapa retomada" )
      "Etapa retomada"()
   END_RUNG
   // the same network as SCL:
   IF "Variaveis"."Etapa pausada" AND NOT "Variaveis"."Etapa retomada" THEN "Etapa pausada"(); END_IF;
   IF NOT "Variaveis"."Etapa pausada" AND "Variaveis"."Etapa retomada" THEN "Etapa retomada"(); END_IF;
END_REGION

REGION Network 5
   RUNG wire#powerrail
      Contact( "Variaveis"."Decisao automatica" )
      Contact( "Variaveis"."Transiciona etapa" )
      wire#w1
      "EB - Etapa finalizada"()
   END_RUNG
   RUNG wire#w1
      R_Coil( "Variaveis"."Realiza EB" )
   END_RUNG
   RUNG wire#w1
      S_Coil( "Variaveis"."Realiza EC" )
   END_RUNG
   RUNG wire#w1
      Coil( "Variaveis"."EC iniciada" )
   END_RUNG
   // the same network as SCL:
   #_w1 := "Variaveis"."Decisao automatica" AND "Variaveis"."Transiciona etapa";
   IF #_w1 THEN
       "EB - Etapa finalizada"();
       "Variaveis"."Realiza EB" := FALSE;
       "Variaveis"."Realiza EC" := TRUE;
   END_IF;
   "Variaveis"."EC iniciada" := #_w1;
END_REGION
END_FUNCTION

FUNCTION "Realiza EC" : Void   // FC38, LAD
{ S7_Optimized_Access := 'TRUE' }
VERSION : 0.1
BEGIN

REGION Network 1
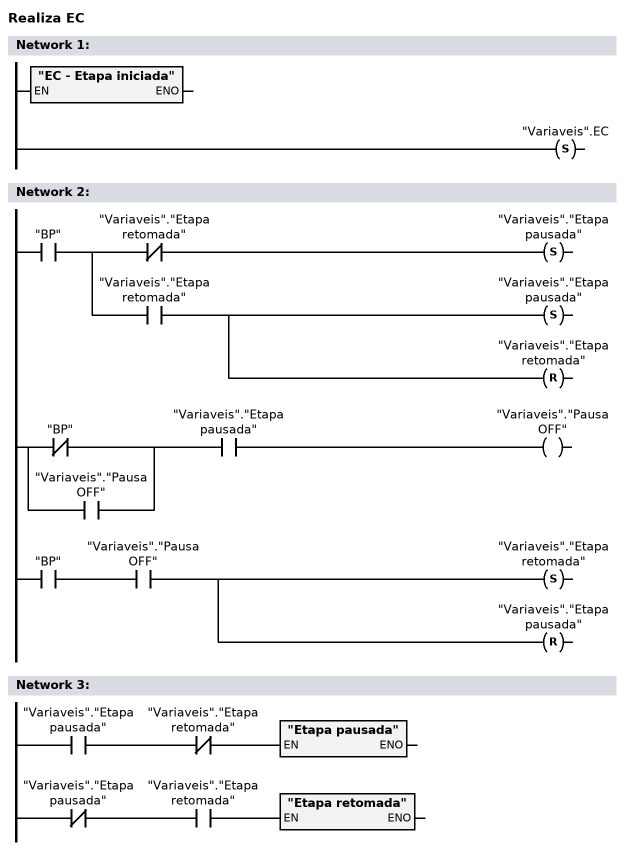
   RUNG wire#powerrail
      "EC - Etapa iniciada"()
   END_RUNG
   RUNG wire#powerrail
      S_Coil( "Variaveis".EC )
   END_RUNG
   // the same network as SCL:
   "EC - Etapa iniciada"();
   "Variaveis".EC := TRUE;
END_REGION

REGION Network 2
   RUNG wire#powerrail
      Contact( "BP" )
      wire#w1
      I_Contact( "Variaveis"."Etapa retomada" )
      S_Coil( "Variaveis"."Etapa pausada" )
   END_RUNG
   RUNG wire#w1
      Contact( "Variaveis"."Etapa retomada" )
      wire#w2
      S_Coil( "Variaveis"."Etapa pausada" )
   END_RUNG
   RUNG wire#w2
      R_Coil( "Variaveis"."Etapa retomada" )
   END_RUNG
   RUNG wire#powerrail
      I_Contact( "BP" )
      wire#w3
      Contact( "Variaveis"."Etapa pausada" )
      Coil( "Variaveis"."Pausa OFF" )
   END_RUNG
   RUNG wire#powerrail
      Contact( "Variaveis"."Pausa OFF" )
   END_RUNG wire#w3
   RUNG wire#powerrail
      Contact( "BP" )
      Contact( "Variaveis"."Pausa OFF" )
      wire#w4
      S_Coil( "Variaveis"."Etapa retomada" )
   END_RUNG
   RUNG wire#w4
      R_Coil( "Variaveis"."Etapa pausada" )
   END_RUNG
   // the same network as SCL:
   IF "BP" AND NOT "Variaveis"."Etapa retomada" THEN "Variaveis"."Etapa pausada" := TRUE; END_IF;
   IF "BP" AND "Variaveis"."Etapa retomada" THEN
       "Variaveis"."Etapa pausada" := TRUE;
       "Variaveis"."Etapa retomada" := FALSE;
   END_IF;
   "Variaveis"."Pausa OFF" := (NOT "BP" OR "Variaveis"."Pausa OFF") AND "Variaveis"."Etapa pausada";
   IF "BP" AND "Variaveis"."Pausa OFF" THEN
       "Variaveis"."Etapa retomada" := TRUE;
       "Variaveis"."Etapa pausada" := FALSE;
   END_IF;
END_REGION

REGION Network 3
   RUNG wire#powerrail
      Contact( "Variaveis"."Etapa pausada" )
      I_Contact( "Variaveis"."Etapa retomada" )
      "Etapa pausada"()
   END_RUNG
   RUNG wire#powerrail
      I_Contact( "Variaveis"."Etapa pausada" )
      Contact( "Variaveis"."Etapa retomada" )
      "Etapa retomada"()
   END_RUNG
   // the same network as SCL:
   IF "Variaveis"."Etapa pausada" AND NOT "Variaveis"."Etapa retomada" THEN "Etapa pausada"(); END_IF;
   IF NOT "Variaveis"."Etapa pausada" AND "Variaveis"."Etapa retomada" THEN "Etapa retomada"(); END_IF;
END_REGION
END_FUNCTION

FUNCTION "MS2 - Operacao finalizada" : Void   // FC39, LAD
{ S7_Optimized_Access := 'TRUE' }
VERSION : 0.1
BEGIN

REGION Network 1
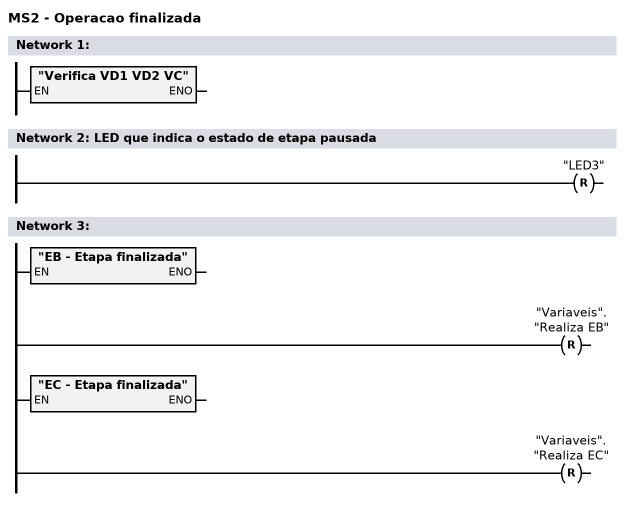
   RUNG wire#powerrail
      "Verifica VD1 VD2 VC"()
   END_RUNG
   // the same network as SCL:
   "Verifica VD1 VD2 VC"();
END_REGION

REGION Network 2: LED que indica o estado de etapa pausada
   RUNG wire#powerrail
      R_Coil( "LED3" )
   END_RUNG
   // the same network as SCL:
   "LED3" := FALSE;
END_REGION

REGION Network 3
   RUNG wire#powerrail
      "EB - Etapa finalizada"()
   END_RUNG
   RUNG wire#powerrail
      R_Coil( "Variaveis"."Realiza EB" )
   END_RUNG
   RUNG wire#powerrail
      "EC - Etapa finalizada"()
   END_RUNG
   RUNG wire#powerrail
      R_Coil( "Variaveis"."Realiza EC" )
   END_RUNG
   // the same network as SCL:
   "EB - Etapa finalizada"();
   "Variaveis"."Realiza EB" := FALSE;
   "EC - Etapa finalizada"();
   "Variaveis"."Realiza EC" := FALSE;
END_REGION
END_FUNCTION

FUNCTION "Verifica VD1 VD2 VC" : Void   // FC40, LAD
{ S7_Optimized_Access := 'TRUE' }
VERSION : 0.1
BEGIN

REGION Network 1: Válvula on/off da entrada do sistema de compressores
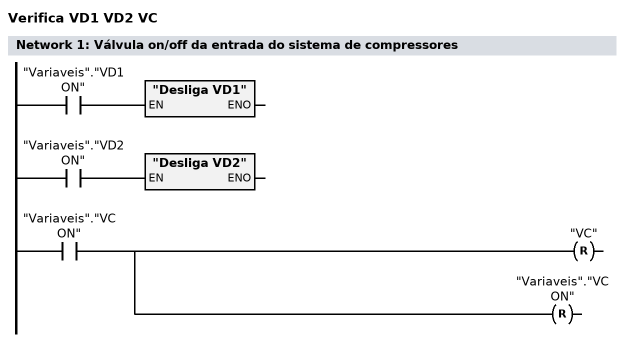
   RUNG wire#powerrail
      Contact( "Variaveis"."VD1 ON" )
      "Desliga VD1"()
   END_RUNG
   RUNG wire#powerrail
      Contact( "Variaveis"."VD2 ON" )
      "Desliga VD2"()
   END_RUNG
   RUNG wire#powerrail
      Contact( "Variaveis"."VC ON" )
      wire#w1
      R_Coil( "VC" )
   END_RUNG
   RUNG wire#w1
      R_Coil( "Variaveis"."VC ON" )
   END_RUNG
   // the same network as SCL:
   IF "Variaveis"."VD1 ON" THEN "Desliga VD1"(); END_IF;
   IF "Variaveis"."VD2 ON" THEN "Desliga VD2"(); END_IF;
   IF "Variaveis"."VC ON" THEN
       "VC" := FALSE;
       "Variaveis"."VC ON" := FALSE;
   END_IF;
END_REGION
END_FUNCTION

FUNCTION "Aciona VD1" : Void   // FC41, LAD
{ S7_Optimized_Access := 'TRUE' }
VERSION : 0.1
BEGIN

REGION Network 1: Válvula on/off da linha direta (primeira)
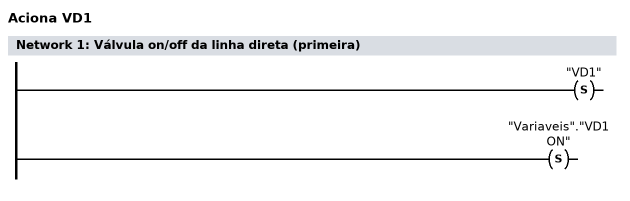
   RUNG wire#powerrail
      S_Coil( "VD1" )
   END_RUNG
   RUNG wire#powerrail
      S_Coil( "Variaveis"."VD1 ON" )
   END_RUNG
   // the same network as SCL:
   "VD1" := TRUE;
   "Variaveis"."VD1 ON" := TRUE;
END_REGION
END_FUNCTION

FUNCTION "Desliga VD1" : Void   // FC42, LAD
{ S7_Optimized_Access := 'TRUE' }
VERSION : 0.1
BEGIN

REGION Network 1: Válvula on/off da linha direta (primeira)
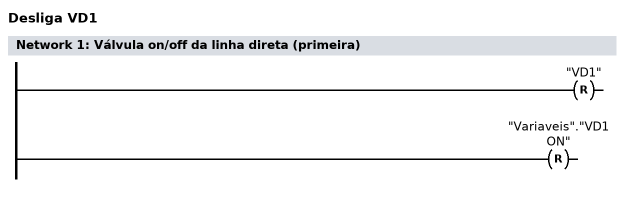
   RUNG wire#powerrail
      R_Coil( "VD1" )
   END_RUNG
   RUNG wire#powerrail
      R_Coil( "Variaveis"."VD1 ON" )
   END_RUNG
   // the same network as SCL:
   "VD1" := FALSE;
   "Variaveis"."VD1 ON" := FALSE;
END_REGION
END_FUNCTION

FUNCTION "OPERACAO - MS2" : Void   // FC43, LAD
{ S7_Optimized_Access := 'TRUE' }
VERSION : 0.1
   VAR_TEMP
      T : Real;   // Temperatura no nó estendido
   END_VAR
   VAR_TEMP   // added for the SCL form of the ladder/FBD networks
      _w1 : Bool;
   END_VAR
BEGIN

REGION Network 1: LED que indica se há alguma operação em curso
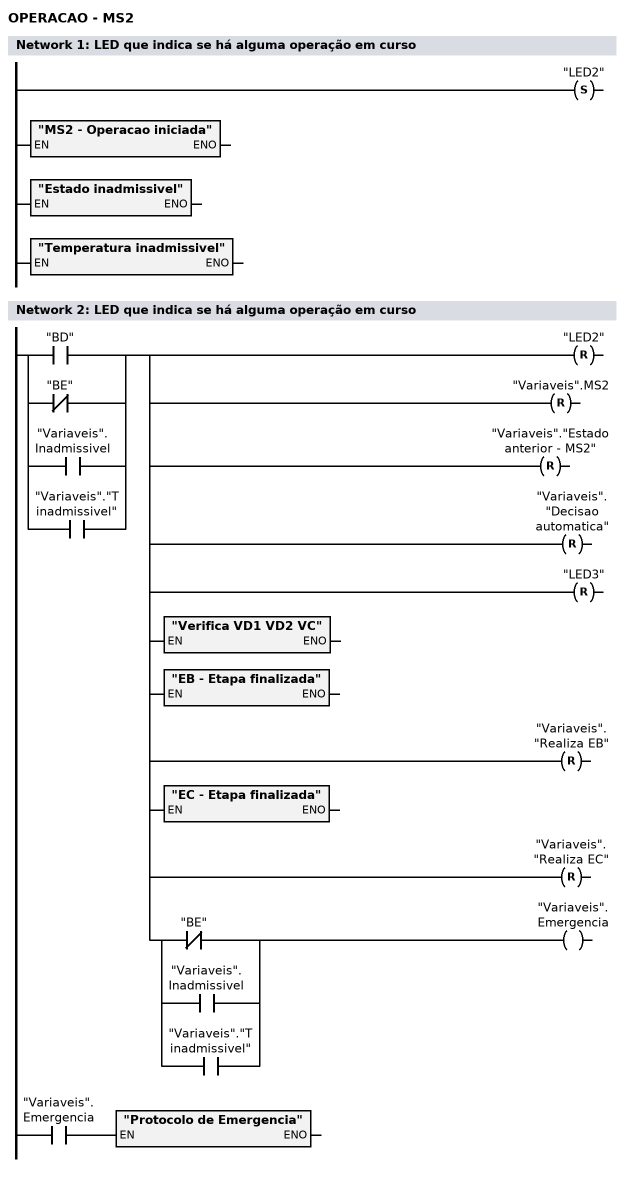
   RUNG wire#powerrail
      S_Coil( "LED2" )
   END_RUNG
   RUNG wire#powerrail
      "MS2 - Operacao iniciada"()
   END_RUNG
   RUNG wire#powerrail
      "Estado inadmissivel"()
   END_RUNG
   RUNG wire#powerrail
      "Temperatura inadmissivel"()
   END_RUNG
   // the same network as SCL:
   "LED2" := TRUE;
   "MS2 - Operacao iniciada"();
   "Estado inadmissivel"();
   "Temperatura inadmissivel"();
END_REGION

REGION Network 2: LED que indica se há alguma operação em curso
   RUNG wire#powerrail
      Contact( "BD" )
      wire#w1
      R_Coil( "LED2" )
   END_RUNG
   RUNG wire#powerrail
      I_Contact( "BE" )
   END_RUNG wire#w1
   RUNG wire#powerrail
      Contact( "Variaveis".Inadmissivel )
   END_RUNG wire#w1
   RUNG wire#powerrail
      Contact( "Variaveis"."T inadmissivel" )
   END_RUNG wire#w1
   RUNG wire#w1
      R_Coil( "Variaveis".MS2 )
   END_RUNG
   RUNG wire#w1
      R_Coil( "Variaveis"."Estado anterior - MS2" )
   END_RUNG
   RUNG wire#w1
      R_Coil( "Variaveis"."Decisao automatica" )
   END_RUNG
   RUNG wire#w1
      R_Coil( "LED3" )
   END_RUNG
   RUNG wire#w1
      "Verifica VD1 VD2 VC"()
   END_RUNG
   RUNG wire#w1
      "EB - Etapa finalizada"()
   END_RUNG
   RUNG wire#w1
      R_Coil( "Variaveis"."Realiza EB" )
   END_RUNG
   RUNG wire#w1
      "EC - Etapa finalizada"()
   END_RUNG
   RUNG wire#w1
      R_Coil( "Variaveis"."Realiza EC" )
   END_RUNG
   RUNG wire#w1
      I_Contact( "BE" )
      wire#w2
      Coil( "Variaveis".Emergencia )
   END_RUNG
   RUNG wire#w1
      Contact( "Variaveis".Inadmissivel )
   END_RUNG wire#w2
   RUNG wire#w1
      Contact( "Variaveis"."T inadmissivel" )
   END_RUNG wire#w2
   RUNG wire#powerrail
      Contact( "Variaveis".Emergencia )
      "Protocolo de Emergencia"()
   END_RUNG
   // the same network as SCL:
   #_w1 := "BD" OR NOT "BE" OR "Variaveis".Inadmissivel OR "Variaveis"."T inadmissivel";
   IF #_w1 THEN
       "LED2" := FALSE;
       "Variaveis".MS2 := FALSE;
       "Variaveis"."Estado anterior - MS2" := FALSE;
       "Variaveis"."Decisao automatica" := FALSE;
       "LED3" := FALSE;
       "Verifica VD1 VD2 VC"();
       "EB - Etapa finalizada"();
       "Variaveis"."Realiza EB" := FALSE;
       "EC - Etapa finalizada"();
       "Variaveis"."Realiza EC" := FALSE;
   END_IF;
   "Variaveis".Emergencia := #_w1 AND (NOT "BE" OR "Variaveis".Inadmissivel OR "Variaveis"."T inadmissivel");
   IF "Variaveis".Emergencia THEN "Protocolo de Emergencia"(); END_IF;
END_REGION
END_FUNCTION

FUNCTION "Temperatura inadmissivel" : Void   // FC44, LAD
{ S7_Optimized_Access := 'TRUE' }
VERSION : 0.1
   VAR_TEMP
      T : Real;   // Temperatura no nó estendido
   END_VAR
BEGIN

REGION Network 1
